PROGRAM MAIN
VAR
	bEnable 		: BOOL;
	bStart  		: BOOL;
	nINT			: INT;
	nUINT			: UINT;
	fREAL			: REAL;
	sPowerStatus	: STRING;
	nFloatConversion : INT;
	fFloatConversion : LREAL;
	nFloatcon2		 : INT;
	fFloatcon2		 : LREAL :=10.1;
END_VAR

bEnable := bStart;

nINT := -32768;
nUINT := 65535;
fREAL := 255.255;

sPowerStatus := 'Power OFF';

fFloatConversion := nFloatConversion;

nFloatcon2 := LREAL_TO_INT(fFloatcon2);

END_PROGRAM

(* stored: Version 1.1.0.1, ProductVersion 3.1.4024.12
   POU MAIN: Id {4d222c44-e74d-4dc9-b8f1-5cd97db1da90}, SpecialFunc None *)
